{attribute 'qualified_only'}
VAR_GLOBAL
	// Mover Velocity
	MoverVelo		: LREAL := 200;
	MoverGap		: LREAL := 180; // Do not exceed 250 mm, or go lower then default
	// Mover Rotation Velocity
	MoverSpinVelo	: LREAL := 1000;
	// Station 2 Mover Index
	Indx			: UDINT;
END_VAR

(* stored: Version 1.1.0.1
   GVL GVL: Id {a162ae6a-45c9-45a0-aa22-1e1fad1763da} *)
